PROGRAM PasosDosificar
VAR_IN_OUT
	iStep:INT;
END_VAR
VAR
	counter:INT;
	dosificando1:BOOL;
	FinDosificado:BOOL;
END_VAR

//Antes de verificar a dosagem, desliga todas as bombas. É preciso para que não fique nenhuma bomba ligada caso o processo pare no meio	
(*FOR counter := 1 TO 12 DO
	Liquidos.InyectarLiq[counter]:=FALSE;
END_FOR
FOR counter := 1 TO 2 DO
	Polvos.InyectarPolvo[counter]:=TRUE	;
END_FOR
*)
CASE iStep OF
	1: counter:=1;
	IF NOT dosificando1 THEN
		FOR counter:=1 TO 12 BY 1 DO
			IF Receta_Activa.SetCircuitosLiq[counter].Paso=iStep THEN
				Liquidos.InyectarLiq[counter]:=TRUE	;
			END_IF
		END_FOR	
		FOR counter:=1 TO 2 BY 1 DO
			IF Receta_Activa.SetCircuitosPo[counter].Paso=iStep THEN
				Polvos.InyectarPolvo[counter]:=TRUE	;
			END_IF
		END_FOR		
	END_IF
	dosificando1:=Liquidos.InyectarLiq[1] OR Liquidos.InyectarLiq[2] OR Liquidos.InyectarLiq[3] OR Liquidos.InyectarLiq[4]OR Liquidos.InyectarLiq[5] OR Liquidos.InyectarLiq[6] OR Liquidos.InyectarLiq[7] OR Liquidos.InyectarLiq[8]OR Liquidos.InyectarLiq[9] OR Liquidos.InyectarLiq[10] OR Liquidos.InyectarLiq[11] OR Liquidos.InyectarLiq[12]OR Polvos.InyectarPolvo[1]OR Polvos.InyectarPolvo[2];
	IF NOT dosificando1 THEN
		iStep:=iStep+1;
	END_IF
	2: counter:=1;
	IF NOT dosificando1 THEN
	FOR counter:=1 TO 12 BY 1 DO
		IF Receta_Activa.SetCircuitosLiq[counter].Paso=iStep THEN
		Liquidos.InyectarLiq[counter]:=TRUE	;
		END_IF
	END_FOR	
	FOR counter:=1 TO 2 BY 1 DO
		IF Receta_Activa.SetCircuitosPo[counter].Paso=iStep THEN
		Polvos.InyectarPolvo[counter]:=TRUE	;
		END_IF
	END_FOR		
	END_IF
	dosificando1:=Liquidos.InyectarLiq[1] OR Liquidos.InyectarLiq[2] OR Liquidos.InyectarLiq[3] OR Liquidos.InyectarLiq[4]OR Liquidos.InyectarLiq[5] OR Liquidos.InyectarLiq[6] OR Liquidos.InyectarLiq[7] OR Liquidos.InyectarLiq[8]OR Liquidos.InyectarLiq[9] OR Liquidos.InyectarLiq[10] OR Liquidos.InyectarLiq[11] OR Liquidos.InyectarLiq[12]OR Polvos.InyectarPolvo[1]OR Polvos.InyectarPolvo[2];
	IF NOT dosificando1 THEN
		iStep:=iStep+1;
	END_IF
	3: counter:=1;
	IF NOT dosificando1 THEN
	FOR counter:=1 TO 12 BY 1 DO
		IF Receta_Activa.SetCircuitosLiq[counter].Paso=iStep THEN
		Liquidos.InyectarLiq[counter]:=TRUE	;
		END_IF
	END_FOR
	FOR counter:=1 TO 2 BY 1 DO
		IF Receta_Activa.SetCircuitosPo[counter].Paso=iStep THEN
		Polvos.InyectarPolvo[counter]:=TRUE	;
		END_IF
	END_FOR			
	END_IF
	dosificando1:=Liquidos.InyectarLiq[1] OR Liquidos.InyectarLiq[2] OR Liquidos.InyectarLiq[3] OR Liquidos.InyectarLiq[4]OR Liquidos.InyectarLiq[5] OR Liquidos.InyectarLiq[6] OR Liquidos.InyectarLiq[7] OR Liquidos.InyectarLiq[8]OR Liquidos.InyectarLiq[9] OR Liquidos.InyectarLiq[10] OR Liquidos.InyectarLiq[11] OR Liquidos.InyectarLiq[12]OR Polvos.InyectarPolvo[1]OR Polvos.InyectarPolvo[2];
	IF NOT dosificando1 THEN
		iStep:=iStep+1;
	END_IF
	4: counter:=1;
	IF NOT dosificando1 THEN
	FOR counter:=1 TO 12 BY 1 DO
		IF Receta_Activa.SetCircuitosLiq[counter].Paso=iStep THEN
		Liquidos.InyectarLiq[counter]:=TRUE	;
		END_IF
	END_FOR
	FOR counter:=1 TO 2 BY 1 DO
		IF Receta_Activa.SetCircuitosPo[counter].Paso=iStep THEN
		Polvos.InyectarPolvo[counter]:=TRUE	;
		END_IF
	END_FOR			
	END_IF
	dosificando1:=Liquidos.InyectarLiq[1] OR Liquidos.InyectarLiq[2] OR Liquidos.InyectarLiq[3] OR Liquidos.InyectarLiq[4]OR Liquidos.InyectarLiq[5] OR Liquidos.InyectarLiq[6] OR Liquidos.InyectarLiq[7] OR Liquidos.InyectarLiq[8]OR Liquidos.InyectarLiq[9] OR Liquidos.InyectarLiq[10] OR Liquidos.InyectarLiq[11] OR Liquidos.InyectarLiq[12]OR Polvos.InyectarPolvo[1]OR Polvos.InyectarPolvo[2];
	IF NOT dosificando1 THEN
		iStep:=iStep+1;
	END_IF
	5: counter:=1;
	IF NOT dosificando1 THEN
	FOR counter:=1 TO 12 BY 1 DO
		IF Receta_Activa.SetCircuitosLiq[counter].Paso=iStep THEN
		Liquidos.InyectarLiq[counter]:=TRUE	;
		END_IF
	END_FOR
	FOR counter:=1 TO 2 BY 1 DO
		IF Receta_Activa.SetCircuitosPo[counter].Paso=iStep THEN
		Polvos.InyectarPolvo[counter]:=TRUE	;
		END_IF
	END_FOR			
	END_IF
	dosificando1:=Liquidos.InyectarLiq[1] OR Liquidos.InyectarLiq[2] OR Liquidos.InyectarLiq[3] OR Liquidos.InyectarLiq[4]OR Liquidos.InyectarLiq[5] OR Liquidos.InyectarLiq[6] OR Liquidos.InyectarLiq[7] OR Liquidos.InyectarLiq[8]OR Liquidos.InyectarLiq[9] OR Liquidos.InyectarLiq[10] OR Liquidos.InyectarLiq[11] OR Liquidos.InyectarLiq[12]OR Polvos.InyectarPolvo[1]OR Polvos.InyectarPolvo[2];
	IF NOT dosificando1 THEN
		iStep:=iStep+1;
	END_IF
	6: counter:=1;
	IF NOT dosificando1 THEN
	FOR counter:=1 TO 12 BY 1 DO
		IF Receta_Activa.SetCircuitosLiq[counter].Paso=iStep THEN
		Liquidos.InyectarLiq[counter]:=TRUE	;
		END_IF
	END_FOR
	FOR counter:=1 TO 2 BY 1 DO
		IF Receta_Activa.SetCircuitosPo[counter].Paso=iStep THEN
		Polvos.InyectarPolvo[counter]:=TRUE	;
		END_IF
	END_FOR			
	END_IF
	dosificando1:=Liquidos.InyectarLiq[1] OR Liquidos.InyectarLiq[2] OR Liquidos.InyectarLiq[3] OR Liquidos.InyectarLiq[4]OR Liquidos.InyectarLiq[5] OR Liquidos.InyectarLiq[6] OR Liquidos.InyectarLiq[7] OR Liquidos.InyectarLiq[8]OR Liquidos.InyectarLiq[9] OR Liquidos.InyectarLiq[10] OR Liquidos.InyectarLiq[11] OR Liquidos.InyectarLiq[12]OR Polvos.InyectarPolvo[1]OR Polvos.InyectarPolvo[2];
	IF NOT dosificando1 THEN
		iStep:=iStep+1;
	END_IF
	7: counter:=1;
	IF NOT dosificando1 THEN
	FOR counter:=1 TO 12 BY 1 DO
		IF Receta_Activa.SetCircuitosLiq[counter].Paso=iStep THEN
		Liquidos.InyectarLiq[counter]:=TRUE	;
		END_IF
	END_FOR
	FOR counter:=1 TO 2 BY 1 DO
		IF Receta_Activa.SetCircuitosPo[counter].Paso=iStep THEN
		Polvos.InyectarPolvo[counter]:=TRUE	;
		END_IF
	END_FOR			
	END_IF
	dosificando1:=Liquidos.InyectarLiq[1] OR Liquidos.InyectarLiq[2] OR Liquidos.InyectarLiq[3] OR Liquidos.InyectarLiq[4]OR Liquidos.InyectarLiq[5] OR Liquidos.InyectarLiq[6] OR Liquidos.InyectarLiq[7] OR Liquidos.InyectarLiq[8]OR Liquidos.InyectarLiq[9] OR Liquidos.InyectarLiq[10] OR Liquidos.InyectarLiq[11] OR Liquidos.InyectarLiq[12]OR Polvos.InyectarPolvo[1]OR Polvos.InyectarPolvo[2];
	IF NOT dosificando1 THEN
		iStep:=iStep+1;
	END_IF
	8: counter:=1;
	IF NOT dosificando1 THEN
		FOR counter:=1 TO 12 BY 1 DO
			IF Receta_Activa.SetCircuitosLiq[counter].Paso=iStep THEN
			Liquidos.InyectarLiq[counter]:=TRUE	;
			END_IF
		END_FOR
		FOR counter:=1 TO 2 BY 1 DO
			IF Receta_Activa.SetCircuitosPo[counter].Paso=iStep THEN
			Polvos.InyectarPolvo[counter]:=TRUE	;
			END_IF
		END_FOR			
	END_IF
	dosificando1:=Liquidos.InyectarLiq[1] OR Liquidos.InyectarLiq[2] OR Liquidos.InyectarLiq[3] OR Liquidos.InyectarLiq[4]OR Liquidos.InyectarLiq[5] OR Liquidos.InyectarLiq[6] OR Liquidos.InyectarLiq[7] OR Liquidos.InyectarLiq[8]OR Liquidos.InyectarLiq[9] OR Liquidos.InyectarLiq[10] OR Liquidos.InyectarLiq[11] OR Liquidos.InyectarLiq[12]OR Polvos.InyectarPolvo[1]OR Polvos.InyectarPolvo[2];
	IF NOT dosificando1 THEN
		iStep:=iStep+1;
	END_IF
	ELSE
		FinDosificado:=TRUE;
END_CASE

END_PROGRAM

(* stored: Version 1.1.0.1, ProductVersion 3.1.4024.14
   POU PasosDosificar: Id {6168d9ce-a74f-4cf5-a967-03cc8af5bcc4}, SpecialFunc None *)
